FUNCTION TIMESTRUCT_TO_DATESTR
VAR_INPUT
  ts: TIMESTRUCT;
END_VAR
VAR_IN_OUT
  outputstr: STRING(255);
END_VAR
VAR
  format_string: FB_FormatString;
END_VAR

format_string(
  sFormat:='%d-%2d-%2d',
  arg1:=F_WORD(ts.wYear),
  arg2:=F_WORD(ts.wMonth),
  arg3:=F_WORD(ts.wDay),
  sOut=>outputstr);

END_FUNCTION

(* stored: Version 1.1.0.1, ProductVersion 3.1.4024.9
   POU TIMESTRUCT_TO_DATESTR: Id {2069b1bd-90ea-4e27-886f-f4662f18b458}, SpecialFunc None *)
